% RSLogix 500 project Automatic_Filler_Wallnuts.RSS, saved by version 8.30.00.16 %
PROJECT "UNTITLED"    % processor: Bul.1763 MicroLogix 1100 Series B %

PROGRAM FILES
  LAD 2 "MAIN"  6 rungs
  LAD 3 "DIGITAL_IO"  8 rungs
  LAD 4 "CONTROLE"  9 rungs
  LAD 5 "ESTADOS"  6 rungs

DATA FILES
  O0 OUTPUT  4 elements
  I1 INPUT  6 elements
  S2 STATUS  66 elements
  B3 BINARY  2 elements
  T4 TIMER  1 elements
  C5 COUNTER  1 elements
  R6 CONTROL  1 elements
  N7 INTEGER  1 elements
  F8 FLOAT  1 elements

LADDER 2 "MAIN"
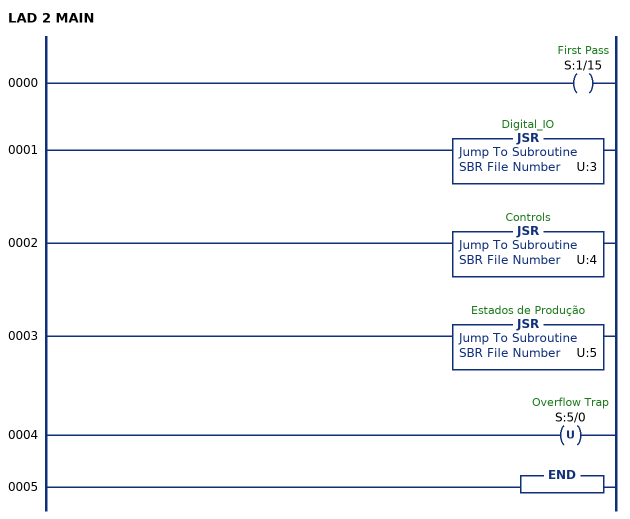
% Rung: 0 %
SOR OTE S:1/15 EOR
%   S:1/15  "First Pass" %
% Rung: 1 %
SOR JSR U:3 EOR
%   U:3  "Digital_IO" %
% Rung: 2 %
SOR JSR U:4 EOR
%   U:4  "Controls" %
% Rung: 3 %
SOR JSR U:5 EOR
%   U:5  "Estados de Produção" %
% Rung: 4 %
SOR OTU S:5/0 EOR
%   S:5/0  "Overflow Trap" %
% Rung: 5 %
SOR END EOR

LADDER 3 "DIGITAL_IO"
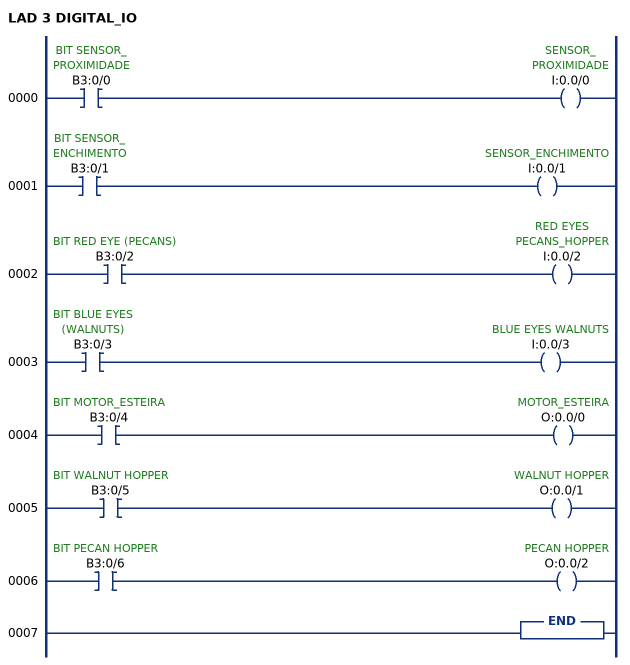
% Rung: 0 %
SOR XIC B3:0/0 OTE I:0.0/0 EOR
%   B3:0/0  "BIT SENSOR_PROXIMIDADE" %
%   I:0.0/0  "SENSOR_PROXIMIDADE" %
% Rung: 1 %
SOR XIC B3:0/1 OTE I:0.0/1 EOR
%   B3:0/1  "BIT SENSOR_ENCHIMENTO" %
%   I:0.0/1  "SENSOR_ENCHIMENTO" %
% Rung: 2 %
SOR XIC B3:0/2 OTE I:0.0/2 EOR
%   B3:0/2  "BIT RED EYE (PECANS)" %
%   I:0.0/2  PECANS_HOPPER  "RED EYES" %
% Rung: 3 %
SOR XIC B3:0/3 OTE I:0.0/3 EOR
%   B3:0/3  "BIT BLUE EYES (WALNUTS)" %
%   I:0.0/3  WALNUTS  "BLUE EYES" %
% Rung: 4 %
SOR XIC B3:0/4 OTE O:0.0/0 EOR
%   B3:0/4  "BIT MOTOR_ESTEIRA" %
%   O:0.0/0  "MOTOR_ESTEIRA" %
% Rung: 5 %
SOR XIC B3:0/5 OTE O:0.0/1 EOR
%   B3:0/5  "BIT WALNUT HOPPER" %
%   O:0.0/1  "WALNUT HOPPER" %
% Rung: 6 %
SOR XIC B3:0/6 OTE O:0.0/2 EOR
%   B3:0/6  "BIT PECAN HOPPER" %
%   O:0.0/2  "PECAN HOPPER" %
% Rung: 7 %
SOR END EOR

LADDER 4 "CONTROLE"
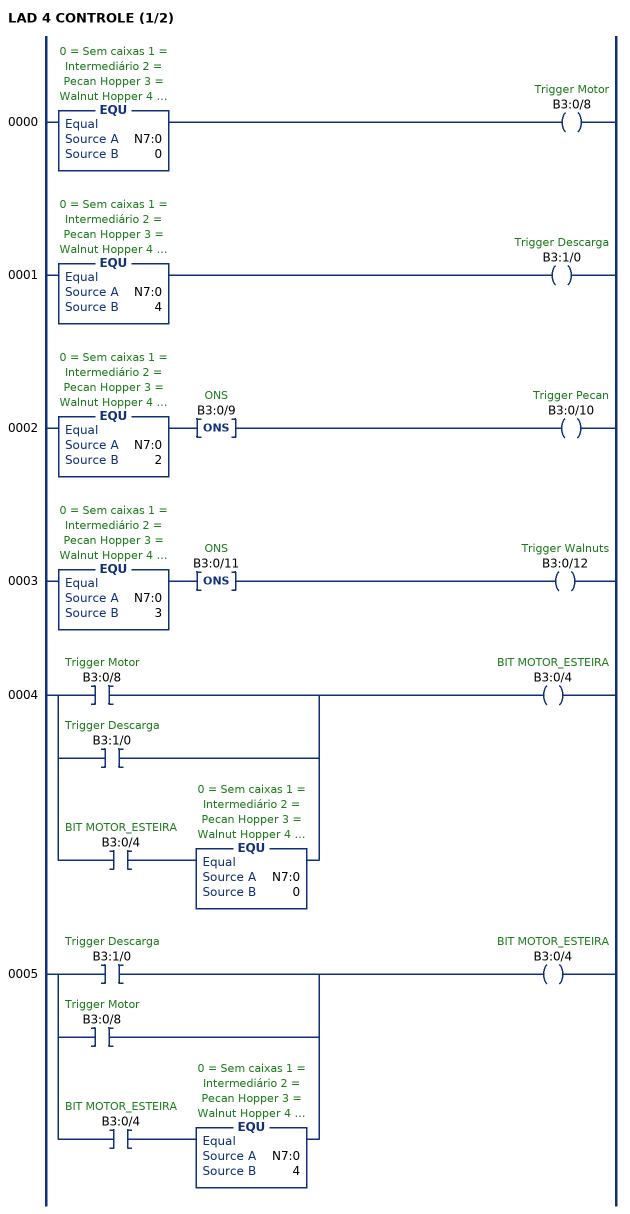
% Rung: 0 %
SOR EQU N7:0 0 OTE B3:0/8 EOR
%   N7:0  "0 = Sem caixas 1 = Intermediário 2 = Pecan Hopper 3 = Walnut Hopper 4 = Descarga de Caix" %
%   B3:0/8  "Trigger Motor" %
% Rung: 1 %
SOR EQU N7:0 4 OTE B3:1/0 EOR
%   N7:0  "0 = Sem caixas 1 = Intermediário 2 = Pecan Hopper 3 = Walnut Hopper 4 = Descarga de Caix" %
%   B3:1/0  "Trigger Descarga" %
% Rung: 2 %
SOR EQU N7:0 2 ONS B3:0/9 OTE B3:0/10 EOR
%   N7:0  "0 = Sem caixas 1 = Intermediário 2 = Pecan Hopper 3 = Walnut Hopper 4 = Descarga de Caix" %
%   B3:0/9  "ONS" %
%   B3:0/10  "Trigger Pecan" %
% Rung: 3 %
SOR EQU N7:0 3 ONS B3:0/11 OTE B3:0/12 EOR
%   N7:0  "0 = Sem caixas 1 = Intermediário 2 = Pecan Hopper 3 = Walnut Hopper 4 = Descarga de Caix" %
%   B3:0/11  "ONS" %
%   B3:0/12  "Trigger Walnuts" %
% Rung: 4 %
SOR BST XIC B3:0/8 NXB XIC B3:1/0 NXB XIC B3:0/4 EQU N7:0 0 BND OTE B3:0/4 EOR
%   B3:0/8  "Trigger Motor" %
%   B3:1/0  "Trigger Descarga" %
%   B3:0/4  "BIT MOTOR_ESTEIRA" %
%   N7:0  "0 = Sem caixas 1 = Intermediário 2 = Pecan Hopper 3 = Walnut Hopper 4 = Descarga de Caix" %
% Rung: 5 %
SOR BST XIC B3:1/0 NXB XIC B3:0/8 NXB XIC B3:0/4 EQU N7:0 4 BND OTE B3:0/4 EOR
%   B3:1/0  "Trigger Descarga" %
%   B3:0/8  "Trigger Motor" %
%   B3:0/4  "BIT MOTOR_ESTEIRA" %
%   N7:0  "0 = Sem caixas 1 = Intermediário 2 = Pecan Hopper 3 = Walnut Hopper 4 = Descarga de Caix" %

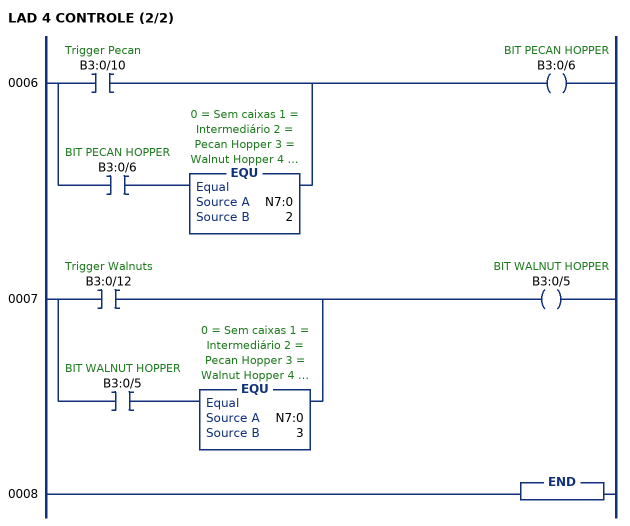
% Rung: 6 %
SOR BST XIC B3:0/10 NXB XIC B3:0/6 EQU N7:0 2 BND OTE B3:0/6 EOR
%   B3:0/10  "Trigger Pecan" %
%   B3:0/6  "BIT PECAN HOPPER" %
%   N7:0  "0 = Sem caixas 1 = Intermediário 2 = Pecan Hopper 3 = Walnut Hopper 4 = Descarga de Caix" %
% Rung: 7 %
SOR BST XIC B3:0/12 NXB XIC B3:0/5 EQU N7:0 3 BND OTE B3:0/5 EOR
%   B3:0/12  "Trigger Walnuts" %
%   B3:0/5  "BIT WALNUT HOPPER" %
%   N7:0  "0 = Sem caixas 1 = Intermediário 2 = Pecan Hopper 3 = Walnut Hopper 4 = Descarga de Caix" %
% Rung: 8 %
SOR END EOR

LADDER 5 "ESTADOS"
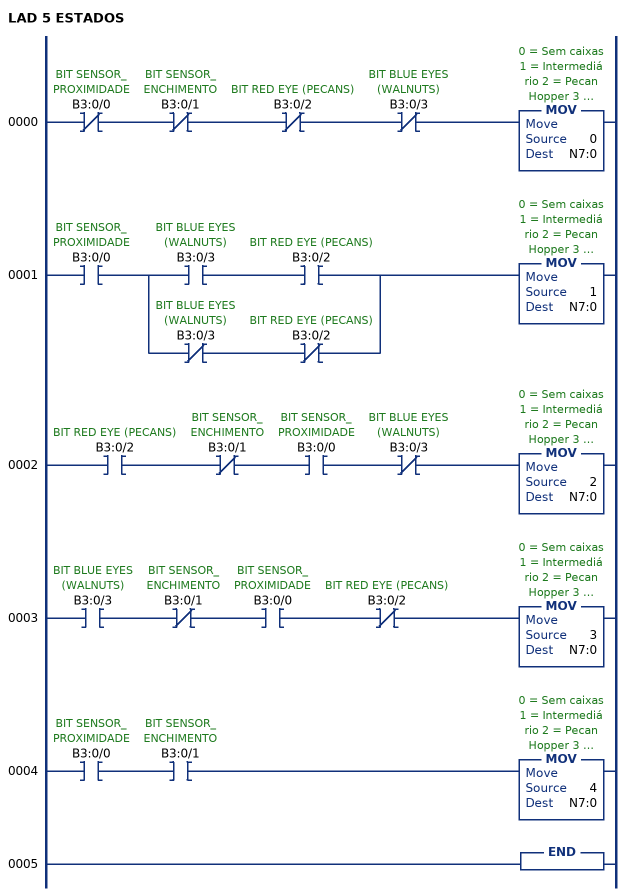
% Rung: 0 %
SOR XIO B3:0/0 XIO B3:0/1 XIO B3:0/2 XIO B3:0/3 MOV 0 N7:0 EOR
%   B3:0/0  "BIT SENSOR_PROXIMIDADE" %
%   B3:0/1  "BIT SENSOR_ENCHIMENTO" %
%   B3:0/2  "BIT RED EYE (PECANS)" %
%   B3:0/3  "BIT BLUE EYES (WALNUTS)" %
%   N7:0  "0 = Sem caixas 1 = Intermediário 2 = Pecan Hopper 3 = Walnut Hopper 4 = Descarga de Caix" %
% Rung: 1 %
SOR XIC B3:0/0 BST XIC B3:0/3 XIC B3:0/2 NXB XIO B3:0/3 XIO B3:0/2 BND MOV 1 N7:0 EOR
%   B3:0/0  "BIT SENSOR_PROXIMIDADE" %
%   B3:0/3  "BIT BLUE EYES (WALNUTS)" %
%   B3:0/2  "BIT RED EYE (PECANS)" %
%   N7:0  "0 = Sem caixas 1 = Intermediário 2 = Pecan Hopper 3 = Walnut Hopper 4 = Descarga de Caix" %
% Rung: 2 %
SOR XIC B3:0/2 XIO B3:0/1 XIC B3:0/0 XIO B3:0/3 MOV 2 N7:0 EOR
%   B3:0/2  "BIT RED EYE (PECANS)" %
%   B3:0/1  "BIT SENSOR_ENCHIMENTO" %
%   B3:0/0  "BIT SENSOR_PROXIMIDADE" %
%   B3:0/3  "BIT BLUE EYES (WALNUTS)" %
%   N7:0  "0 = Sem caixas 1 = Intermediário 2 = Pecan Hopper 3 = Walnut Hopper 4 = Descarga de Caix" %
% Rung: 3 %
SOR XIC B3:0/3 XIO B3:0/1 XIC B3:0/0 XIO B3:0/2 MOV 3 N7:0 EOR
%   B3:0/3  "BIT BLUE EYES (WALNUTS)" %
%   B3:0/1  "BIT SENSOR_ENCHIMENTO" %
%   B3:0/0  "BIT SENSOR_PROXIMIDADE" %
%   B3:0/2  "BIT RED EYE (PECANS)" %
%   N7:0  "0 = Sem caixas 1 = Intermediário 2 = Pecan Hopper 3 = Walnut Hopper 4 = Descarga de Caix" %
% Rung: 4 %
SOR XIC B3:0/0 XIC B3:0/1 MOV 4 N7:0 EOR
%   B3:0/0  "BIT SENSOR_PROXIMIDADE" %
%   B3:0/1  "BIT SENSOR_ENCHIMENTO" %
%   N7:0  "0 = Sem caixas 1 = Intermediário 2 = Pecan Hopper 3 = Walnut Hopper 4 = Descarga de Caix" %
% Rung: 5 %
SOR END EOR

OTHER DOCUMENTED ADDRESSES
  B3:0/7  "One SHOT"
  B3:0/13  "ONS"
  B3:0/14  "Trigger Descarga"

DATA TABLE (non-zero values as saved)
DATA B3
% B3:0 % 0X011C 0X0000
